{attribute addProperty BoxType "KL9160"}
{attribute addProperty Id "Channel_1Channel_0970199100"}
{attribute addProperty CRC "2629167143"}
{attribute addProperty SizeInBites "0"}
{attribute addProperty SizeInBytes "0"}
TYPE KL9160_9CB5E827 :
STRUCT
	{attribute addProperty Name "Channel_1"}
	Channel_1 : Channel_09701991;
END_STRUCT
END_TYPE

(* stored: Version 1.2.0.0, ProductVersion 3.1.4024.9
   DUT KL9160_9CB5E827: Id {e6522c74-fa8a-4a4c-b1f1-af56b1d19d73} *)
